// TwinCAT 3 PLC project PRG_MachineControl_HMI_Connector
// Title: B_MachineControl_HMI_Connector
// Company: RafalOS
// Author: Rafal Osajda
// ProjectVersion: 0.0.0.3
// ProgramVersion: 3.1.4024.0
// libraries:
//   B_Base, * (RafalOS)
//   B_Base_HMI_Connector, * (RafalOS)
//   B_HMIElements, * (RafalOS)
//   B_MachineControl, * (RafalOS)
//   B_StatesAndModes, * (RafalOS)
//   Tc2_Standard, * (Beckhoff Automation GmbH)
//   Tc2_System, * (Beckhoff Automation GmbH)
//   Tc3_Module, * (Beckhoff Automation GmbH)
// project tree:
//   / PlcTask.TcTTO
//   POUs Compilation/ PRGCompilation.TcPOU (not stored)
//   POUs/01_MC/ FB_MCHMIMachineControl_HMI.TcPOU, ITF_MCHMIMachineControl_HMI.TcIO (not stored), ST_MCHMIMachineControl_HMI_Link.TcDUT, ST_MCHMIMachineControl_HMI.TcDUT (not stored)
//   POUs/02_RodzicDlaPrzygotowywanieStron/ FB_MCHMIPrepareDataForScreen.TcPOU, ITF_MCHMIPrepareDataForScreen.TcIO (not stored)
// real-time tasks:
//   TASK PlcTask: cycle T#10ms, priority 20, ADS port 350

CONFIGURATION PRG_MachineControl_HMI_Connector
    RESOURCE PLC ON TwinCAT3
        TASK PlcTask(INTERVAL := T#10ms, PRIORITY := 20);
        PROGRAM PRGCompilation WITH PlcTask : PRGCompilation;
    END_RESOURCE
END_CONFIGURATION

// ---- POUs/01_MC/ST_MCHMIMachineControl_HMI_Link.TcDUT
TYPE ST_MCHMIMachineControl_HMI_Link EXTENDS ST_BaseTopElement_HMI_Link :
STRUCT
	stMachineControl		: ST_MCHMIMachineControl_HMI;
END_STRUCT
END_TYPE

// ---- POUs/01_MC/FB_MCHMIMachineControl_HMI.TcPOU
FUNCTION_BLOCK FB_MCHMIMachineControl_HMI EXTENDS FB_BaseTopElement_HMI IMPLEMENTS ITF_MCHMIMachineControl_HMI
VAR
	itfMachineControlConnector			: ITF_MCMachineControl_HMI_Connector;
	refstMachineControlData				: REFERENCE TO ST_MCHMIMachineControl_HMI;
	(*	Przygotowywanie danych dla ramek	*)
	arrPrepareScreen					: ARRAY [0..GVL_HMIEConstans.MAX_NUMBER_OF_BUTTON_IN_MENU] OF 
											ARRAY [0..GVL_SaMConstans.NUMBER_OF_MODES] OF ITF_MCHMIPrepareDataForScreen;
END_VAR

METHOD PUBLIC AddPrepareScreenModuleFromManager : BOOL
VAR_INPUT
END_VAR
END_METHOD

(*			
	RafalOS
	Rafał Osajda		19.11.2025		TC 4024.66
	Sprzątanie po stronie wywoływane z HMIManager i wywołująca odpowiednią metode z ITF z arrPrepareScreen
*)
METHOD ClearAfterScreenFroHMIManager : BOOL
VAR_INPUT
	iScreen		: INT;
	iMode		: INT;
END_VAR
END_METHOD

METHOD FB_init : BOOL
VAR_INPUT
	bInitRetains : BOOL; // if TRUE, the retain variables are initialized (warm start / cold start)
	bInCopyCode : BOOL;  // if TRUE, the instance afterwards gets moved into the copy code (online change)
	itfBaseLoggerConnector				: ITF_BaseLogger_HMI_Connector;	//bezpośredni łącznik do logera
	itfMachineControlConnector			: ITF_MCMachineControl_HMI_Connector;
END_VAR
//Przypisanie do elementu który własnie stworzyliśmy
THIS^.itfMachineControlConnector := itfMachineControlConnector;
//Przypisanie do elementów z biblioteki
THIS^.itfBaseLoggerElementConnector := itfMachineControlConnector;
THIS^.itfBaseComponentConnector := itfMachineControlConnector;
THIS^.itfBaseControlElementConnector := itfMachineControlConnector;
THIS^.itfBaseGroupElementConnector := itfMachineControlConnector;
THIS^.itfBaseTopElementConnector := itfMachineControlConnector;
//
THIS^.itfBaseLoggerConnector := itfBaseLoggerConnector;

IF (THIS^.itfMachineControlConnector <> 0 AND
	THIS^.itfBaseLoggerElementConnector <> 0 AND
	THIS^.itfBaseComponentConnector	<> 0 AND
	THIS^.itfBaseControlElementConnector <> 0 AND
	THIS^.itfBaseGroupElementConnector <> 0 AND
	THIS^.itfBaseTopElementConnector <> 0 AND
	THIS^.itfBaseLoggerConnector <> 0) THEN
	THIS^.bIsInit						:= TRUE;
END_IF
END_METHOD

METHOD PUBLIC LinkMachineControlData : BOOL
VAR_INPUT
	stData			: REFERENCE TO ST_MCHMIMachineControl_HMI_Link;
END_VAR
THIS^.refstMachineControlData REF= stData.stMachineControl;

THIS^.refstBaseLoggerElementDataHMI REF= stData.stBaseLoggerElement;
THIS^.refstBaseComponentDataHMI REF= stData.stBaseComponent;
THIS^.refstBaseControlElementDataHMI REF= stData.stBaseControlElement;
THIS^.refstBaseGroupElementDataHMI REF= stData.stBaseGroupElement;
THIS^.refstBaseTopElementDataHMI REF= stData.stBaseTopElement;

THIS^.CreateLinkToEventsMemory ();

IF (__ISVALIDREF (THIS^.refstMachineControlData) AND THIS^.IsLinkedReferences ()) THEN
	THIS^.bIsValidData := TRUE;
	LinkMachineControlData := TRUE;
END_IF
END_METHOD

(*			
	RafalOS
	Rafał Osajda		19.11.2025		TC 4024.66
	Przygotowanie danych dla strony wywoływane z HMIManager i wywołująca odpowiednią metode z ITF z arrPrepareScreen
*)
METHOD PrepareDataForScreenFromHMIManager : BOOL
VAR_INPUT
	iScreen		: INT;
	iMode		: INT;
END_VAR
END_METHOD

(*			
	RafalOS
	Rafał Osajda		19.11.2025		TC 4024.66
	Przygotowanie strony wywoływane z HMIManager i wywołująca odpowiednią metode z ITF z arrPrepareScreen
*)
METHOD PrepareForScreenFromHMIManager : BOOL
VAR_INPUT
	iScreen		: INT;
	iMode		: INT;
END_VAR
END_METHOD

END_FUNCTION_BLOCK

// ---- POUs/02_RodzicDlaPrzygotowywanieStron/FB_MCHMIPrepareDataForScreen.TcPOU
(*			
	RafalOS
	Rafał Osajda		19.11.2025		TC 4024.66
	Domyślne przygotowanie danych dla ekranu
*)
FUNCTION_BLOCK FB_MCHMIPrepareDataForScreen EXTENDS FB_BaseComponent_HMI IMPLEMENTS ITF_MCHMIMachineControl_HMI
VAR
	//itf do lacznika machinecontrol
	//strulture danych 
	//dodać ITF dla możliwości obsługi rozszerzonej obsługi wyświetlania 
END_VAR

(*			
	RafalOS
	Rafał Osajda		19.11.2025		TC 4024.66
	Czyści danych przy zmienia ramki po poprzedniej ramce
*)
METHOD PUBLIC ClearAfterScreen : BOOL
VAR_INPUT
END_VAR
SUPER^.ClearAfterScreen ();
END_METHOD

(*			
	RafalOS
	Rafał Osajda		14.11.2025		TC 4024.66
	Metoda przygotowywania danych dla HMI 
	W niej odbywa się odpytywanie właściego elementu przez łącznik
*)
METHOD PUBLIC PrepareDataForHMI : BOOL
VAR_INPUT
END_VAR
SUPER^.PrepareDataForHMI ();
END_METHOD

(*			
	RafalOS
	Rafał Osajda		19.11.2025		TC 4024.66
	Przygotowanie ramki pood tamke do wyświetlenia - tylko przygotowanie a nie przygotowanie danych do wyświetlenia
*)
METHOD PUBLIC PrepareForScreen : BOOL
VAR_INPUT
END_VAR
SUPER^.PrepareForScreen ();
END_METHOD

END_FUNCTION_BLOCK
